// TIA Portal V18 export
// export: Created 2026-01-09T11:31:53.8816638Z, ExportSetting WithDefaults, DisplayName Totally Integrated Automation Portal, DisplayVersion V18 Update 5, DisplayName TIA Portal Openness, DisplayVersion V18 Update 5, DisplayName TIA Portal Teamcenter Gateway, DisplayVersion V18, DisplayName TIA Portal Version Control Interface, DisplayVersion V18, DisplayName SINAMICS Startdrive Advanced, DisplayVersion V18 SP2 Update 1, DisplayName SINAMICS Startdrive G110M, G120, G120C, G120D, G120P, G115D, DisplayVersion V18 SP2 Update 1, DisplayName SINAMICS Startdrive G130, G150, S120, S150, SINAMICS MV, S210, G220, S200, DisplayVersion V18 SP2 Update 1, DisplayName STEP 7 Professional, DisplayVersion V18 Update 5, DisplayName STEP 7 Safety, DisplayVersion V18, DisplayName WinCC Professional, DisplayVersion V18 Update 5
TagTable "Pallet"
  AutoProcessControl_Global_H_EmptyPallet : Bool  (PLC tag AutoProcessControl.Global.H.EmptyPallet, CPU S71500-2PN_TP700, 100 ms)
  AutoProcessControl_Global_J_EmptyPallet : Bool  (PLC tag AutoProcessControl.Global.J.EmptyPallet, CPU S71500-2PN_TP700, 100 ms)
  AutoProcessControl_Global_K_EmptyPallet : Bool  (PLC tag AutoProcessControl.Global.K.EmptyPallet, CPU S71500-2PN_TP700, 100 ms)
  AutoProcessControl_Global_L_EmptyPallet : Bool  (PLC tag AutoProcessControl.Global.L.EmptyPallet, CPU S71500-2PN_TP700, 100 ms)
  AutoProcessControl_Global_ALL_EmptyPallet : Bool  (PLC tag AutoProcessControl.Global.ALL_EmptyPallet, CPU S71500-2PN_TP700, 100 ms)
  AutoProcessControl_Robot_3_PalletFull(1) : Bool  (PLC tag AutoProcessControl.Robot_3.PalletFull, CPU S71500-2PN_TP700, 1 s)
